INTERFACE iTrack

PROPERTY CurrentMoverCount : DINT
GET
END_GET
END_PROPERTY

PROPERTY CurrentMoverList : iMoverList
GET
END_GET
END_PROPERTY

PROPERTY Id : INT
GET
END_GET
SET
END_SET
END_PROPERTY

METHOD RegisterMover : BOOL
VAR_INPUT
    NewMover : REFERENCE TO Mover;
END_VAR
VAR
END_VAR
END_METHOD

METHOD UnregisterAll : BOOL
VAR_INPUT
END_VAR
END_METHOD

METHOD UnregisterMover : BOOL
VAR_INPUT
    RemovingMover : REFERENCE TO Mover;
END_VAR
VAR
END_VAR
END_METHOD

END_INTERFACE

(* stored: Version 1.1.0.1, ProductVersion 3.1.4024.12
   Itf iTrack: Id {41e6f11d-1951-01da-13f4-8ac69ce6b873}
   Folder Methods: Id {cc616af7-fa5e-0721-3c8e-d062b484e0c8}
   Folder Properties: Id {332f2434-e8e7-012d-221e-b1241870310e}
   Property CurrentMoverCount: Id {7706471b-0127-0e08-2769-e211435d9cd2}
   Get Get: Id {f904841d-fff0-0874-075a-461b289a34a3}
   Property CurrentMoverList: Id {53b54c82-4385-0644-3c7a-fe140dee0acc}
   Get Get: Id {f55b5545-5b8d-060b-31cd-65f766a1eda0}
   Property Id: Id {e69e0034-eced-090a-3e7c-cb98c2c8ba20}
   Get Get: Id {fda8bdc8-fe34-01b4-33d1-6cb2adf3c8b1}
   Set Set: Id {eedf83fb-7109-04ab-2166-7221f61f50a7}
   Method RegisterMover: Id {aa379151-5a94-0a15-244b-4ddcbf268ca8}
   Method UnregisterAll: Id {f2ab22b3-a027-08df-22f2-7e3232cd47f0}
   Method UnregisterMover: Id {c8d25a54-3401-08fd-3ce2-76cee9dd2344} *)
